				IF tonExecute.Q THEN
					eCycleState								:= E_ProcessCycle.WAIT_STATION1_MOV1;	
				END_IF

E_ProcessCycle.WAIT_STATION1_MOV1:
				
				IF B_1_1_PRG_Master_Station_1.STATUS.bDone THEN
					eCycleState								:= E_ProcessCycle.STATION2_MOV2;
					stStation1.Mov1							:= FALSE;
					B_1_1_PRG_Master_Station_1.CMD.bExecute	:= FALSE;
					B_1_1_PRG_Master_Station_1.CMD.bReady 	:= TRUE;
				END_IF

E_ProcessCycle.STATION2_MOV2:

				B_1_1_PRG_Master_Station_1.CMD.bReady 		:= FALSE;
				
				stStation2.Mov2								:= TRUE;
				B_2_1_PRG_Master_Station_2.CMD.bExecute		:= TRUE;
				
				IF tonExecute.Q THEN
					eCycleState								:= E_ProcessCycle.WAIT_STATION2_MOV2;	
				END_IF

E_ProcessCycle.WAIT_STATION2_MOV2:

				IF B_2_1_PRG_Master_Station_2.STATUS.bDone THEN
					stStation2.Mov2							:= FALSE;
					B_2_1_PRG_Master_Station_2.CMD.bExecute	:= FALSE;
					B_2_1_PRG_Master_Station_2.CMD.bReady 	:= TRUE;	
					eCycleState								:= E_ProcessCycle.STATION1_MOV3_STATION2_MOV2;
				END_IF

E_ProcessCycle.STATION1_MOV3_STATION2_MOV2:

				B_2_1_PRG_Master_Station_2.CMD.bReady 		:= FALSE;
	
				stStation1.Mov3								:= TRUE;
				stStation2.Mov2								:= TRUE;
				B_2_1_PRG_Master_Station_2.CMD.bExecute		:= TRUE;
				B_1_1_PRG_Master_Station_1.CMD.bExecute		:= TRUE;
				
				IF tonExecute.Q THEN
					eCycleState								:= E_ProcessCycle.WAIT_STATION1_MOV3_STATION2_MOV2;	
				END_IF

E_ProcessCycle.WAIT_STATION1_MOV3_STATION2_MOV2:
			
				IF B_2_1_PRG_Master_Station_2.STATUS.bDone AND B_1_1_PRG_Master_Station_1.STATUS.bDone THEN
					stStation1.Mov3							:= FALSE;
					stStation2.Mov2							:= FALSE;
					B_2_1_PRG_Master_Station_2.CMD.bExecute	:= FALSE;
					B_1_1_PRG_Master_Station_1.CMD.bExecute	:= FALSE;	
					B_2_1_PRG_Master_Station_2.CMD.bReady 	:= TRUE;
					B_1_1_PRG_Master_Station_1.CMD.bReady 	:= TRUE;
					eCycleState								:= E_ProcessCycle.STATION3_MOV3;
				END_IF	

E_ProcessCycle.STATION3_MOV3:

					B_2_1_PRG_Master_Station_2.CMD.bReady 	:= FALSE;
					B_1_1_PRG_Master_Station_1.CMD.bReady 	:= FALSE;
					
					B_3_1_PRG_Master_Station_3.CMD.bExecute	:= TRUE;
					stStation3.Mov3							:= TRUE;
					
				IF tonExecute.Q THEN
					eCycleState								:= E_ProcessCycle.WAIT_STATION3_MOV3;	
				END_IF

E_ProcessCycle.WAIT_STATION3_MOV3:

				IF B_3_1_PRG_Master_Station_3.STATUS.bDone THEN
					stStation3.Mov3							:= FALSE;
					B_3_1_PRG_Master_Station_3.CMD.bExecute	:= FALSE;
					B_3_1_PRG_Master_Station_3.CMD.bReady 	:= TRUE;	
					bIndexDataHistoryFlag					:= TRUE;
					eCycleState								:= E_ProcessCycle.SAVE_DATA;
				END_IF

E_ProcessCycle.SAVE_DATA:

				FOR i := 199 TO 0 BY -1 DO
					aDataHistory[i+1] 						:= aDataHistory[i];
				END_FOR			
				eCycleState									:= E_ProcessCycle.SAVE_DATA2;
					
E_ProcessCycle.SAVE_DATA2:	
				
				c_ACT_SaveData();
				IF tonSave_Data.Q THEN
					eCycleState								:= E_ProcessCycle.CSV;
				END_IF	
				
				
E_ProcessCycle.CSV:
			
				stCSVProcess.bWriteData						:= TRUE;
				IF tonWriteToCsv.Q THEN
					stCSVProcess.bWriteData					:= FALSE;
				END_IF
				IF NOT stCSVProcess.bBusy AND tonWriteToCsv.Q THEN
					eCycleState								:= E_ProcessCycle.RESET_ALL_CMD;
					nIndexDataHistory						:= nIndexDataHistory +1;
				END_IF
				
END_CASE
END_ACTION

ACTION c_ACT_SaveData:
(*rIndexDataHistoryFlag( CLK := 	bIndexDataHistoryFlag);
	IF rIndexDataHistoryFlag.Q THEN
					nIndexDataHistory						:= nIndexDataHistory + 1;
					bIndexDataHistoryFlag					:= FALSE;
	END_IF*)

				
	//STATION 1
	aDataHistory[0].sSetting1_1	:= stCycleDataStation1.sSetting1;
	aDataHistory[0].nSetting2_1	:= stCycleDataStation1.nSetting2;
	aDataHistory[0].bSetting3_1	:= stCycleDataStation1.bSetting3;
	
	aDataHistory[0].sDATA1_1	:= stCycleDataStation1.sDATA1;
	aDataHistory[0].nDATA2_1	:= stCycleDataStation1.nDATA2;
	aDataHistory[0].bDATA3_1	:= stCycleDataStation1.bDATA3;
	
	aDataHistory[0].bPass_1		:= stCycleDataStation1.bPass;
	aDataHistory[0].bFail_1		:= stCycleDataStation1.bFail;
	
	//STATION 2
	aDataHistory[0].sSetting1_2	:= stCycleDataStation2.sSetting1;
	aDataHistory[0].nSetting2_2	:= stCycleDataStation2.nSetting2;
	aDataHistory[0].bSetting3_2	:= stCycleDataStation2.bSetting3;
	
	aDataHistory[0].sDATA1_2	:= stCycleDataStation2.sDATA1;
	aDataHistory[0].nDATA2_2	:= stCycleDataStation2.nDATA2;
	aDataHistory[0].bDATA3_2	:= stCycleDataStation2.bDATA3;
	
	aDataHistory[0].bPass_2		:= stCycleDataStation2.bPass;
	aDataHistory[0].bFail_2		:= stCycleDataStation2.bFail;
	
	//STATION 3
	aDataHistory[0].sSetting1_3	:= stCycleDataStation3.sSetting1;
	aDataHistory[0].nSetting2_3	:= stCycleDataStation3.nSetting2;
	aDataHistory[0].bSetting3_3	:= stCycleDataStation3.bSetting3;
	
	aDataHistory[0].sDATA1_3	:= stCycleDataStation3.sDATA1;
	aDataHistory[0].nDATA2_3	:= stCycleDataStation3.nDATA2;
	aDataHistory[0].bDATA3_3	:= stCycleDataStation3.bDATA3;
	
	aDataHistory[0].bPass_3		:= stCycleDataStation3.bPass;
	aDataHistory[0].bFail_3		:= stCycleDataStation3.bFail;
 
	
	
	aDataHistory[0].bPass		:= bPASS;
	aDataHistory[0].bFail		:= bFAIL;
	aDataHistory[0].sData		:= sSystemDate;
	aDataHistory[0].sTime		:= sSystemTime;
END_ACTION

END_PROGRAM

// ---- POUs/MAIN.TcPOU
PROGRAM MAIN
VAR
END_VAR

A_1_PRG_Main_Master();

END_PROGRAM

// ---- POUs/Utilities/FB_TerminalInfo.TcPOU
FUNCTION_BLOCK FB_TerminalInfo
VAR_INPUT
	 nTerminalState  : UINT;
END_VAR
VAR_OUTPUT
	 sTerminalState  : STRING;
END_VAR
VAR
END_VAR

IF nTerminalState = 1 THEN 
   sTerminalState := 'Initialization';
ELSIF  nTerminalState = 2 THEN 
   sTerminalState := 'PREOP';  
ELSIF  nTerminalState = 3 THEN 
   sTerminalState := 'BOOT'; 
ELSIF  nTerminalState = 4 THEN 
   sTerminalState := 'SAFEOP';   
ELSIF  nTerminalState = 8 THEN 
   sTerminalState := 'OPERATIONAL';
ELSIF  nTerminalState = 16#0010 THEN 
   sTerminalState := 'Slave signals error';   
ELSIF  nTerminalState = 16#0020 THEN 
   sTerminalState := 'Invalid vendorId, productCode... read';  
ELSIF  nTerminalState = 16#0040 THEN 
   sTerminalState := 'Initialization error occurred';   
ELSIF  nTerminalState = 16#0080 THEN 
   sTerminalState := 'Slave disabled';   
ELSIF  nTerminalState = 16#0100 THEN 
   sTerminalState := 'Slave not present';    
ELSIF  nTerminalState = 16#0200 THEN 
   sTerminalState := 'Slave signals link error';    
ELSIF  nTerminalState = 16#0400 THEN 
   sTerminalState := 'Slave signals missing link'; 
ELSIF  nTerminalState = 16#0800 THEN 
   sTerminalState := 'Slave signals unexpected link';
ELSIF  nTerminalState = 16#1000 THEN 
   sTerminalState := 'Communication port A';
ELSIF  nTerminalState = 16#2000 THEN 
   sTerminalState := 'Communication port B';
ELSIF  nTerminalState = 16#4000 THEN 
   sTerminalState := 'Communication port C';
ELSIF  nTerminalState = 16#8000 THEN 
   sTerminalState := 'Communication port D'; 	
END_IF

END_FUNCTION_BLOCK

// ---- POUs/Utilities/FB_TimeControl.TcPOU
FUNCTION_BLOCK PUBLIC FB_TimeControl
VAR_INPUT
	bEnable         :BOOL;
	bReset          :BOOL;
END_VAR
VAR_OUTPUT 
	nHour           :DINT;
	nMin            :DINT;
	nSec            :DINT;
	nTotalSec       :DINT;
END_VAR
VAR
	tpPulse1        :TP;
	tpPulse2        :TP;
	
	
    bMainStart      :BOOL;
    bStart1         :BOOL;
    bStart2         :BOOL;
    bStop           :BOOL;
    bPuls1          :BOOL;
    bPuls2          :BOOL;

    ftrigPuls1      :F_TRIG;
    ftrigPuls2      :F_TRIG;
    rtrigPulsMain   :R_TRIG;
	
	
END_VAR

rtrigPulsMain(CLK:= bEnable);
ftrigPuls1(CLK:= bPuls2);
ftrigPuls2(CLK:= bPuls1);

tpPulse1(IN:=(ftrigPuls1.Q OR rtrigPulsMain.Q) ,PT:= T#490MS);
bPuls1:= tpPulse1.Q;

tpPulse2(IN:=(ftrigPuls2.Q AND NOT bStop) ,PT:= T#490MS);
bPuls2:=tpPulse2.Q;

IF bEnable THEN
	bMainStart := TRUE;
ELSE 
	bMainStart := FALSE;
END_IF
bStop := NOT bMainStart;

IF bMainStart AND ftrigPuls1.Q THEN
	nTotalSec := nTotalSec + 1;
ELSIF bReset THEN
	nTotalSec := 0;
END_IF
//Secend
IF bMainStart AND ftrigPuls1.Q THEN
	nSec := nSec + 1;
	ELSIF (nSec = 60) THEN
	nSec := 0;
	ELSIF bReset THEN
	nSec := 0;	
END_IF
//Minutes
IF bMainStart THEN
	nMin := (nTotalSec-(nHour*3600)) /60;
	ELSIF bReset THEN
	nMin := 0;
END_IF
//Hours
IF bMainStart THEN
	nHour := nTotalSec/3600;
	ELSIF bReset THEN
	nHour := 0;
END_IF

END_FUNCTION_BLOCK
